{attribute 'qualified_only'}
{attribute 'strict'}
TYPE eTcoTixonFeedingSimpleTests :
(
    Restore := 1,
    CleanUp,
    Message,
    PowerDisable,
    PowerEnable,
    Reset,

	
    Last
);
END_TYPE

(* stored: Version 1.1.0.1, ProductVersion 3.1.4024.12
   DUT eTcoTixonFeedingSimpleTests: Id {47a1ee63-9ac0-0c59-0555-13932492fb51} *)
